PROGRAM MAIN
VAR
	myDebug : BOOL;
	ChangeTo1 : BOOL;
	ChangeTo2 : BOOL;
END_VAR

IF myFanControl.IsOn THEN
	myDebug := TRUE;
ELSE 
	myDebug := FALSE;
END_IF

IF ChangeTo1 THEN
	ChangeTo1 := FALSE;
	myFanControlDigitalInput.ChangeDigitalInput(device1.GetDigitalInput(0));
END_IF

IF ChangeTo2 THEN
	ChangeTo2 := FALSE;
	myFanControlDigitalInput.ChangeDigitalInput(device1.GetDigitalInput(1));
END_IF

END_PROGRAM

(* stored: Version 1.1.0.1, ProductVersion 3.1.4024.5
   POU MAIN: Id {6b9cda75-2e94-42d4-8a7f-4c0c520828d2}, SpecialFunc None *)
